// TIA Portal V16 export
// export: Created 2023-03-03T13:43:34.171212Z, ExportSetting WithDefaults, DisplayName Totally Integrated Automation Portal, DisplayVersion V16 Update 3, DisplayName TIA Portal Version Control Interface, DisplayVersion V16 Update 2, DisplayName TIA Portal Openness, DisplayVersion V16 Update 3, DisplayName STEP 7 Professional, DisplayVersion V16 Update 3, DisplayName STEP 7 Safety, DisplayVersion V16, DisplayName WinCC Professional, DisplayVersion V16 Update 3
TYPE "UT39511_Dy_DebugInst1Order"
TITLE = Dynamic UDT [DEBUG] — First Order Response Simulation
// PRACTICAL SERIES AUTOMATION LIBRARY (PAL)   —   COPYRIGHT 2020 – M. GLEDHILL (MIT LICENCE)
//                   ———— ◆ ————
// FULL ONLINE DOCUMENTATION IS AVAILABLE AT: https://practicalseries.com/2001-pal/index.html
// stored: IsFailsafeCompliant false
   STRUCT
      revInfo { ExternalWritable := 'False'} : "UT01000_St_SysRevision";   // ▀▀▀▀ UDT CURRENT REVISION
      ___________0010_0 { ExternalAccessible := 'False'; ExternalVisible := 'False'; ExternalWritable := 'False'} : Int;
      ___________0010_1 { ExternalAccessible := 'False'; ExternalVisible := 'False'; ExternalWritable := 'False'} : Int;   // ▀▀▀▀ CALCULATION CONSTANTS
      k_Gain : Real := 1.0;   // CONSTANT — Simulation system gain
      k_TimeConstant : Real := 1.0;   // CONSTANT — Simulation system time constant (s)
      ___________0020_0 { ExternalAccessible := 'False'; ExternalVisible := 'False'; ExternalWritable := 'False'} : Int;
      ___________0020_1 { ExternalAccessible := 'False'; ExternalVisible := 'False'; ExternalWritable := 'False'} : Int;   // ▀▀▀▀ SIMULATION STATUS SIGNALS
      status_Running : Bool;   // STATUS — Simulation is running (1 = running, 0 = stopped)
      status_Stopped : Bool;   // STATUS — Simulation is stopped (not running) (1 = stopped, 0 = running)
      status_SteadyState : Bool;   // STATUS — Steady state (±2%) achieved (1 = In steady state, 0 = not steady state)
      status_Aut : Bool;   // STATUS — Simulation is in automatic mode (1 = automatic, 0 = manual)
      status_Man : Bool;   // STATUS — Simulation is in manual mode (1 = manual, 0 = automatic)
      ___________0030_0 { ExternalAccessible := 'False'; ExternalVisible := 'False'; ExternalWritable := 'False'} : Int;
      ___________0030_1 { ExternalAccessible := 'False'; ExternalVisible := 'False'; ExternalWritable := 'False'} : Int;   // ▀▀▀▀ CALCULATED VALUES
      cal_TimeSteady : Real;   // CALC — Time to reach steady state, zero for unstable response (s)
      ___________0040_0 { ExternalAccessible := 'False'; ExternalVisible := 'False'; ExternalWritable := 'False'} : Int;
      ___________0040_1 { ExternalAccessible := 'False'; ExternalVisible := 'False'; ExternalWritable := 'False'} : Int;   // ▀▀▀▀ OPERATING MODE SELECTION
      mode_AutMan : Bool := true;   // MODE — Automatic/manual mode selection (1 = auto mode, 0 = manual mode)
      mode_ManTime : Real;   // MODE — Manual mode time value (s)
      ___________0050_0 { ExternalAccessible := 'False'; ExternalVisible := 'False'; ExternalWritable := 'False'} : Int;
      ___________0050_1 { ExternalAccessible := 'False'; ExternalVisible := 'False'; ExternalWritable := 'False'} : Int;   // ▀▀▀▀ LIVE TIMING DATA
      actual_Output : Real;   // ACTUAL — SIMULATION OUTPUT VALUE (identical to OUTPUT parameter)
      actual_PrevOutput : Real;   // ACTUAL — Output value from the previous iteration y[n-1]
      actual_StartTime : DTL;   // ACTUAL — CPU time when simulation started
      actual_Time : DTL;   // ACTUAL — CPU time of this (current) iteration of the calculation
      actual_PrevTime : DTL;   // ACTUAL — CPU time of the previous iteration of the calculation
      actual_RunTime : Real;   // ACTUAL — Elapsed time since the simulation started (s)
      actual_DeltaTime : Real;   // ACTUAL — Time period between this and previous iteration (s)
   END_STRUCT;
   // revInfo.REV_BLOCK := 'UT39511';
   // revInfo.REV_NUMBER := '001.000';
   // revInfo.REV_DATE := '2023-03-03';
   // revInfo.REV_AUTHOR := 'M. Gledhill';
END_TYPE
